(* IEC 61131-3 sources: ICSQuartz/benchmarks/oscat_basic_is_cc/src, 1 file *)

(* ---- program.st ---- *)
PROGRAM PLC_PRG
VAR_INPUT
    in_STR: STRING;
    in_CMP: STRING;
END_VAR

IS_CC(in_STR, in_CMP);

END_PROGRAM
